{attribute 'pack_mode' := '1'} 
// ------------------------------------------------------------------------- 
//  SRCI Robot Library                                                
// ------------------------------------------------------------------------- 
//                                                                           
//  Object:      CalculateCartesianPositionParCmd                                       
//  Author:      Thorsten Brach                                                
//  Date:        2024-06-05
//
//  Description:                                              
//   
//                                                                           
//  Copyright: 
//    (C) 2024 Thorsten Brach. All rights reserved                                                                                                                                            
//             Licensed under the MIT License.
//                                                                           
//  Disclaimer:                                                                           
//    This project is provided without any guarantee and can be used for   
//    private and commercial purposes. Any use is at the user’s 
//    own risk and responsibility.
//
// -------------------------------------------------------------------------
TYPE CalculateCartesianPositionParCmd :
STRUCT
  /// Index of initial frame
  /// • 0: WCS (default)
  /// • 1..254: User frames
  FrameNo            : USINT;
  /// Index of target frame
  /// • 0: WCS (default)
  /// • 1..254: User frames
  TargetFrameNo      : USINT;  
  /// Robot cartesian position.
  CartesianPosition  : RobotCartesianPosition;
END_STRUCT
END_TYPE

{attribute 'pack_mode' := '1'} 
// ------------------------------------------------------------------------- 
//  SRCI Robot Library                                                
// ------------------------------------------------------------------------- 
//                                                                           
//  Object:      CalculateCartesianPositionRecvData                                       
//  Author:      Thorsten Brach                                                
//  Date:        2024-06-05
//
//  Description:                                              
//   
//                                                                           
//  Copyright: 
//    (C) 2024 Thorsten Brach. All rights reserved                                                                                                                                            
//             Licensed under the MIT License.
//                                                                           
//  Disclaimer:                                                                           
//    This project is provided without any guarantee and can be used for   
//    private and commercial purposes. Any use is at the user’s 
//    own risk and responsibility.
//
// -------------------------------------------------------------------------
TYPE CalculateCartesianPositionRecvData EXTENDS RspHeader :
STRUCT
  /// Index of target tool
  /// • 0: Flange (default)
  /// • 1..254: Tool frames
  TargetToolNoReturn       : USINT;
  /// Index of target frame
  /// •      0: WCS
  /// • 1..254: User frames
  TargetFrameNoReturn      : USINT;
  /// Calculated cartesian position
  CartesianPositionReturn  : RobotCartesianPosition;
END_STRUCT
END_TYPE

{attribute 'pack_mode' := '1'}
// ------------------------------------------------------------------------- 
//  SRCI Robot Library                                                
// ------------------------------------------------------------------------- 
//                                                                           
//  Object:      CalculateCartesianPositionSendData                                       
//  Author:      Thorsten Brach                                                
//  Date:        2024-06-05
//
//  Description:                                              
//   
//                                                                           
//  Copyright: 
//    (C) 2024 Thorsten Brach. All rights reserved                                                                                                                                            
//             Licensed under the MIT License.
//                                                                           
//  Disclaimer:                                                                           
//    This project is provided without any guarantee and can be used for   
//    private and commercial purposes. Any use is at the user’s 
//    own risk and responsibility.
//
// -------------------------------------------------------------------------
TYPE CalculateCartesianPositionSendData EXTENDS CmdHeader:   
STRUCT
  /// Index of source frame
  /// • 0: WCS (default)
  /// • 1..254: User frames
  FrameNo           : USINT;
  /// Index of target frame
  /// • 0: WCS (default)
  /// • 1..254: User frames
  TargetFrameNo     : USINT;
  /// Robot cartesian position.
  CartesianPosition : RobotCartesianPosition;
END_STRUCT
END_TYPE

{attribute 'pack_mode' := '1'} 
// ------------------------------------------------------------------------- 
//  SRCI Robot Library                                                
// ------------------------------------------------------------------------- 
//                                                                           
//  Object:      CalculateForwardKinematicOutCmd                                       
//  Author:      Thorsten Brach                                                
//  Date:        2024-06-05
//
//  Description:                                              
//   
//                                                                           
//  Copyright: 
//    (C) 2024 Thorsten Brach. All rights reserved                                                                                                                                            
//             Licensed under the MIT License.
//                                                                           
//  Disclaimer:                                                                           
//    This project is provided without any guarantee and can be used for   
//    private and commercial purposes. Any use is at the user’s 
//    own risk and responsibility.
//
// -------------------------------------------------------------------------
TYPE CalculateForwardKinematicOutCmd :
STRUCT
  /// Index of target tool
  /// • 0: Flange (default)
  /// • 1..254: Tool frames
  TargetToolNoReturn : USINT;
  /// Index of target frame
  /// •      0: WCS
  /// • 1..254: User frames
  TargetFrameNoReturn: USINT;
  /// Calculated cartesian position
  CartesianPosition  : RobotCartesianPosition;
END_STRUCT
END_TYPE

{attribute 'pack_mode' := '1'} 
// ------------------------------------------------------------------------- 
//  SRCI Robot Library                                                
// ------------------------------------------------------------------------- 
//                                                                           
//  Object:      CalculateForwardKinematicParCmd                                       
//  Author:      Thorsten Brach                                                
//  Date:        2024-06-05
//
//  Description:                                              
//   
//                                                                           
//  Copyright: 
//    (C) 2024 Thorsten Brach. All rights reserved                                                                                                                                            
//             Licensed under the MIT License.
//                                                                           
//  Disclaimer:                                                                           
//    This project is provided without any guarantee and can be used for   
//    private and commercial purposes. Any use is at the user’s 
//    own risk and responsibility.
//
// -------------------------------------------------------------------------
TYPE CalculateForwardKinematicParCmd :
STRUCT
  /// Index of target tool
  /// • 0: Flange (default)
  /// • 1..254: Tool frames
  ToolNo             : USINT;
  /// Index of target frame
  /// • 0: WCS (default)
  /// • 1..254: User frames
  FrameNo            : USINT;
  /// Calculate joint position
  JointPosition      : RobotJointPosition;
END_STRUCT
END_TYPE

{attribute 'pack_mode' := '1'} 
// ------------------------------------------------------------------------- 
//  SRCI Robot Library                                                
// ------------------------------------------------------------------------- 
//                                                                           
//  Object:      CalculateForwardKinematicRecvData                                       
//  Author:      Thorsten Brach                                                
//  Date:        2024-06-05
//
//  Description:                                              
//   
//                                                                           
//  Copyright: 
//    (C) 2024 Thorsten Brach. All rights reserved                                                                                                                                            
//             Licensed under the MIT License.
//                                                                           
//  Disclaimer:                                                                           
//    This project is provided without any guarantee and can be used for   
//    private and commercial purposes. Any use is at the user’s 
//    own risk and responsibility.
//
// -------------------------------------------------------------------------
TYPE CalculateForwardKinematicRecvData EXTENDS RspHeader :
STRUCT
  /// Index of target tool
  /// • 0: Flange (default)
  /// • 1..254: Tool frames
  TargetToolNoReturn       : USINT;
  /// Index of target frame
  /// •      0: WCS
  /// • 1..254: User frames
  TargetFrameNoReturn      : USINT;
  /// Calculated cartesian position
  CartesianPosition        : RobotCartesianPosition;
END_STRUCT
END_TYPE

{attribute 'pack_mode' := '1'}
// ------------------------------------------------------------------------- 
//  SRCI Robot Library                                                
// ------------------------------------------------------------------------- 
//                                                                           
//  Object:      CalculateForwardKinematicSendData                                       
//  Author:      Thorsten Brach                                                
//  Date:        2024-06-05
//
//  Description:                                              
//   
//                                                                           
//  Copyright: 
//    (C) 2024 Thorsten Brach. All rights reserved                                                                                                                                            
//             Licensed under the MIT License.
//                                                                           
//  Disclaimer:                                                                           
//    This project is provided without any guarantee and can be used for   
//    private and commercial purposes. Any use is at the user’s 
//    own risk and responsibility.
//
// -------------------------------------------------------------------------
TYPE CalculateForwardKinematicSendData EXTENDS CmdHeader:   
STRUCT
  /// Index of target tool
  /// • 0: Flange (default)
  /// • 1..254: Tool frames
  ToolNo        : USINT;
  /// Index of target frame
  /// • 0: WCS (default)
  /// • 1..254: User frames
  FrameNo        : USINT;
  /// Calculated joint position
  JointPosition  : RobotJointPosition;
END_STRUCT
END_TYPE

{attribute 'pack_mode' := '1'} 
// ------------------------------------------------------------------------- 
//  SRCI Robot Library                                                
// ------------------------------------------------------------------------- 
//                                                                           
//  Object:      CalculateFrameOutCmd                                       
//  Author:      Thorsten Brach                                                
//  Date:        2024-06-09
//
//  Description:                                              
//   
//                                                                           
//  Copyright: 
//    (C) 2024 Thorsten Brach. All rights reserved                                                                                                                                            
//             Licensed under the MIT License.
//                                                                           
//  Disclaimer:                                                                           
//    This project is provided without any guarantee and can be used for   
//    private and commercial purposes. Any use is at the user’s 
//    own risk and responsibility.
//
// -------------------------------------------------------------------------
TYPE CalculateFrameOutCmd :
STRUCT
  /// Date
  IEC_Date       : IEC_DATE;
  /// Time
  IEC_TIME       : IEC_TIME;
  /// Index of frame on which the calculated frame is depending
  /// •      0: WCS (default)
  /// • 1..254: User frames
  ReferenceFrame : USINT;
  /// Position
  Position       : RobotCartesianPositionBase;
END_STRUCT
END_TYPE

{attribute 'pack_mode' := '1'} 
// ------------------------------------------------------------------------- 
//  SRCI Robot Library                                                
// ------------------------------------------------------------------------- 
//                                                                           
//  Object:      CalculateFrameParCmd                                       
//  Author:      Thorsten Brach                                                
//  Date:        2024-06-09
//
//  Description:                                              
//   
//                                                                           
//  Copyright: 
//    (C) 2024 Thorsten Brach. All rights reserved                                                                                                                                            
//             Licensed under the MIT License.
//                                                                           
//  Disclaimer:                                                                           
//    This project is provided without any guarantee and can be used for   
//    private and commercial purposes. Any use is at the user’s 
//    own risk and responsibility.
//
// -------------------------------------------------------------------------
TYPE CalculateFrameParCmd :
STRUCT
  /// Define which method should be used to calculate the tool frame
  Mode               : FrameCalculationMode;
  /// Index of target frame
  /// • 0: WCS (default)
  /// • 1..254: User frames
  FrameNo            : USINT;  
  /// Cartesian position in the positive direction of the  X-Axis of the calculated frame coordinate system relative to the given frame
  Position_X         : RobotCartesianPosition;
  /// Cartesian position in the XY-plane of the calculated frame coordinate system relative to the given frame.
  Position_XY        : RobotCartesianPosition;
  /// Cartesian position of the origin of the calculated frame coordinate system relative to the given frame.
  Origin             : RobotCartesianPosition;
  /// Cartesian position of the postponement of the origin of the calculated frame coordinate system relative to the given frame.
  /// Auxiliary position if the origin of the can’t be reached by the robot, i.e. because it is inside an object.
  OriginShift        : RobotCartesianPosition;
  /// Index of frame on which the calculated frame is depending
  /// •      0: WCS (default)
  /// • 1..254: User frames
  ReferenceFrame     : USINT;
END_STRUCT
END_TYPE

{attribute 'pack_mode' := '1'} 
// ------------------------------------------------------------------------- 
//  SRCI Robot Library                                                
// ------------------------------------------------------------------------- 
//                                                                           
//  Object:      CalculateFrameRecvData                                       
//  Author:      Thorsten Brach                                                
//  Date:        2024-06-09
//
//  Description:                                              
//   
//                                                                           
//  Copyright: 
//    (C) 2024 Thorsten Brach. All rights reserved                                                                                                                                            
//             Licensed under the MIT License.
//                                                                           
//  Disclaimer:                                                                           
//    This project is provided without any guarantee and can be used for   
//    private and commercial purposes. Any use is at the user’s 
//    own risk and responsibility.
//
// -------------------------------------------------------------------------
TYPE CalculateFrameRecvData EXTENDS RspHeader :
STRUCT
  /// Date
  IEC_Date       : IEC_DATE;
  /// Time
  IEC_TIME       : IEC_TIME;
  /// Index of frame on which the calculated frame is depending
  /// •      0: WCS (default)
  /// • 1..254: User frames
  ReferenceFrame : USINT;
  /// Reserve
  Reserve        : BYTE;
  /// Position
  Position       : RobotCartesianPositionBase;
END_STRUCT
END_TYPE

{attribute 'pack_mode' := '1'}
// ------------------------------------------------------------------------- 
//  SRCI Robot Library                                                
// ------------------------------------------------------------------------- 
//                                                                           
//  Object:      CalculateFrameSendData                                       
//  Author:      Thorsten Brach                                                
//  Date:        2024-06-09
//
//  Description:                                              
//   
//                                                                           
//  Copyright: 
//    (C) 2024 Thorsten Brach. All rights reserved                                                                                                                                            
//             Licensed under the MIT License.
//                                                                           
//  Disclaimer:                                                                           
//    This project is provided without any guarantee and can be used for   
//    private and commercial purposes. Any use is at the user’s 
//    own risk and responsibility.
//
// -------------------------------------------------------------------------
TYPE CalculateFrameSendData EXTENDS CmdHeader:   
STRUCT
  /// Incremented with each position of the input parameter "PositionsArray" sent from the PLC to the RC.
  /// Default: 0
  DataIndex          : USINT;
  
  /// Set TRUE by the client, when according to the user selected "Mode" the final position of the input parameter "PositionsArray" is sent to the RC.
  /// Default: FALSE
  DataComplete       : BYTE;
  ///
  Reserve            : BYTE;
  /// Index of target frame
  /// • 0: WCS (default)
  /// • 1..254: User frames
  FrameNo            : USINT;
  /// Index of frame on which the calculated frame is depending
  /// •      0: WCS (default)
  /// • 1..254: User frames
  ReferenceFrame     : USINT;
  /// Define which method should be used to calculate the frame coordinate system: M
  /// • 0: Three-Point-Method (default) O
  /// • 1: Four-Point-Method O
  /// • 2: One-Point-Method
  Mode               : SINT;  
  /// Cartesian position
  Position           : RobotCartesianPosition;  
END_STRUCT
END_TYPE

{attribute 'pack_mode' := '1'} 
// ------------------------------------------------------------------------- 
//  SRCI Robot Library                                                
// ------------------------------------------------------------------------- 
//                                                                           
//  Object:      CalculateInverseKinematicOutCmd                                       
//  Author:      Thorsten Brach                                                
//  Date:        2024-06-09
//
//  Description:                                              
//   
//                                                                           
//  Copyright: 
//    (C) 2024 Thorsten Brach. All rights reserved                                                                                                                                                                                                               
//             Licensed under the MIT License.
//                                                                           
//  Disclaimer:                                                                           
//    This project is provided without any guarantee and can be used for   
//    private and commercial purposes. Any use is at the user’s 
//    own risk and responsibility.
//
// -------------------------------------------------------------------------
TYPE CalculateInverseKinematicOutCmd :
STRUCT
  /// Calculated robot joint position
  JointPosition      : RobotJointPosition;  
END_STRUCT
END_TYPE

{attribute 'pack_mode' := '1'} 
// ------------------------------------------------------------------------- 
//  SRCI Robot Library                                                
// ------------------------------------------------------------------------- 
//                                                                           
//  Object:      CalculateInverseKinematicParCmd                                       
//  Author:      Thorsten Brach                                                
//  Date:        2024-06-09
//
//  Description:                                              
//   
//                                                                           
//  Copyright: 
//    (C) 2024 Thorsten Brach. All rights reserved                                                                                                                                      
//             Licensed under the MIT License.
//                                                                           
//  Disclaimer:                                                                           
//    This project is provided without any guarantee and can be used for   
//    private and commercial purposes. Any use is at the user’s 
//    own risk and responsibility.
//
// -------------------------------------------------------------------------
TYPE CalculateInverseKinematicParCmd :
STRUCT
  /// cartesian position
  CartesianPosition  : RobotCartesianPosition;
  /// Index of target tool
  /// • 0: Flange (default)
  /// • 1..254: Tool frames
  ToolNo             : USINT;
  /// Index of target frame
  /// • 0: WCS (default)
  /// • 1..254: User frames
  FrameNo            : USINT;  
END_STRUCT
END_TYPE

{attribute 'pack_mode' := '1'} 
// ------------------------------------------------------------------------- 
//  SRCI Robot Library                                                
// ------------------------------------------------------------------------- 
//                                                                           
//  Object:      CalculateInverseKinematicRecvData                                       
//  Author:      Thorsten Brach                                                
//  Date:        2024-06-09
//
//  Description:                                              
//   
//                                                                           
//  Copyright: 
//    (C) 2024 Thorsten Brach. All rights reserved                                                                                                                                            
//             Licensed under the MIT License.
//                                                                           
//  Disclaimer:                                                                           
//    This project is provided without any guarantee and can be used for   
//    private and commercial purposes. Any use is at the user’s 
//    own risk and responsibility.
//
// -------------------------------------------------------------------------
TYPE CalculateInverseKinematicRecvData EXTENDS RspHeader :
STRUCT
  /// Calculated robot joint position
  JointPosition      : RobotJointPosition;  
END_STRUCT
END_TYPE

{attribute 'pack_mode' := '1'}
// ------------------------------------------------------------------------- 
//  SRCI Robot Library                                                
// ------------------------------------------------------------------------- 
//                                                                           
//  Object:      CalculateInverseKinematicSendData                                       
//  Author:      Thorsten Brach                                                
//  Date:        2024-06-09
//
//  Description:                                              
//   
//                                                                           
//  Copyright: 
//    (C) 2024 Thorsten Brach. All rights reserved                                                                                                                                            
//             Licensed under the MIT License.
//                                                                           
//  Disclaimer:                                                                           
//    This project is provided without any guarantee and can be used for   
//    private and commercial purposes. Any use is at the user’s 
//    own risk and responsibility.
//
// -------------------------------------------------------------------------
TYPE CalculateInverseKinematicSendData EXTENDS CmdHeader:   
STRUCT
  /// cartesian position
  CartesianPosition  : RobotCartesianPosition;
  /// Index of target tool
  /// • 0: Flange (default)
  /// • 1..254: Tool frames
  ToolNo             : USINT;
  /// Index of target frame
  /// • 0: WCS (default)
  /// • 1..254: User frames
  FrameNo            : USINT;  
END_STRUCT
END_TYPE

{attribute 'pack_mode' := '1'} 
// ------------------------------------------------------------------------- 
//  SRCI Robot Library                                                
// ------------------------------------------------------------------------- 
//                                                                           
//  Object:      CalculateToolOutCmd                                       
//  Author:      Thorsten Brach                                                
//  Date:        2024-06-09
//
//  Description:                                              
//   
//                                                                           
//  Copyright: 
//    (C) 2024 Thorsten Brach. All rights reserved                                                                                                                                                                                                               
//             Licensed under the MIT License.
//                                                                           
//  Disclaimer:                                                                           
//    This project is provided without any guarantee and can be used for   
//    private and commercial purposes. Any use is at the user’s 
//    own risk and responsibility.
//
// -------------------------------------------------------------------------
TYPE CalculateToolOutCmd :
STRUCT
  /// Tool data
  ToolData           : ToolData;
  /// Maximum error of deviation of the TCP position
  /// from the fix point in world coordinate system
  /// If not supported: • -1
  TCPMaxError       : REAL;
  /// Average error of TCP position from the fix point  in world coordinate system
  /// If not supported: • -1 
  TCPMeanError      : REAL;
END_STRUCT
END_TYPE

{attribute 'pack_mode' := '1'} 
// ------------------------------------------------------------------------- 
//  SRCI Robot Library                                                
// ------------------------------------------------------------------------- 
//                                                                           
//  Object:      CalculateToolParCmd                                       
//  Author:      Thorsten Brach                                                
//  Date:        2024-06-09
//
//  Description:                                              
//   
//                                                                           
//  Copyright: 
//    (C) 2024 Thorsten Brach. All rights reserved                                                                                                                                      
//             Licensed under the MIT License.
//                                                                           
//  Disclaimer:                                                                           
//    This project is provided without any guarantee and can be used for   
//    private and commercial purposes. Any use is at the user’s 
//    own risk and responsibility.
//
// -------------------------------------------------------------------------
TYPE CalculateToolParCmd :
STRUCT
  /// Define which method should be used to calculate the tool frame
  Mode               : ToolCalculationMode;
  /// Index of target tool
  /// • 0: Flange (default)
  /// • 1..254: Tool frames
  ToolNo             : USINT;
  /// Index of target frame
  /// • 0: WCS (default)
  /// • 1..254: User frames
  FrameNo            : USINT;  
  /// • True: Tool fixed
  /// • False: Tool on flange (default)
  ExternalTCP        : BOOL;
  /// Positions in cartesian coordinates for the tool frame calculation.
  PositionsArray     : ARRAY[0..5] OF RobotCartesianPosition;
END_STRUCT
END_TYPE

{attribute 'pack_mode' := '1'} 
// ------------------------------------------------------------------------- 
//  SRCI Robot Library                                                
// ------------------------------------------------------------------------- 
//                                                                           
//  Object:      CalculateToolRecvData                                       
//  Author:      Thorsten Brach                                                
//  Date:        2024-06-09
//
//  Description:                                              
//   
//                                                                           
//  Copyright: 
//    (C) 2024 Thorsten Brach. All rights reserved                                                                                                                                            
//             Licensed under the MIT License.
//                                                                           
//  Disclaimer:                                                                           
//    This project is provided without any guarantee and can be used for   
//    private and commercial purposes. Any use is at the user’s 
//    own risk and responsibility.
//
// -------------------------------------------------------------------------
TYPE CalculateToolRecvData EXTENDS RspHeader :
STRUCT
  /// Maximum error of deviation of the TCP position
  /// from the fix point in world coordinate system
  /// If not supported: • -1
  TCPMaxError       : REAL;
  /// Average error of TCP position from the fix point  in world coordinate system
  /// If not supported: • -1 
  TCPMeanError      : REAL;
  /// Tool data
  ToolData           : ToolData;
END_STRUCT
END_TYPE

{attribute 'pack_mode' := '1'}
// ------------------------------------------------------------------------- 
//  SRCI Robot Library                                                
// ------------------------------------------------------------------------- 
//                                                                           
//  Object:      CalculateToolSendData                                       
//  Author:      Thorsten Brach                                                
//  Date:        2024-06-09
//
//  Description:                                              
//   
//                                                                           
//  Copyright: 
//    (C) 2024 Thorsten Brach. All rights reserved                                                                                                                                            
//             Licensed under the MIT License.
//                                                                           
//  Disclaimer:                                                                           
//    This project is provided without any guarantee and can be used for   
//    private and commercial purposes. Any use is at the user’s 
//    own risk and responsibility.
//
// -------------------------------------------------------------------------
TYPE CalculateToolSendData EXTENDS CmdHeader:   
STRUCT
  DataIndex    : USINT;
  ///
  DataComplete : BYTE;
  /// Index of target tool
  /// • 0: Flange (default)
  /// • 1..254: Tool frames
  ToolNo       : USINT;
  /// Index of target frame
  /// • 0: WCS (default)
  /// • 1..254: User frames
  FrameNo      : USINT;    
  /// Define which method should be used to calculate the tool frame
  Mode         : ToolCalculationMode;
  /// • True: Tool fixed
  /// • False: Tool on flange (default)
  ExternalTCP  : USINT;
  /// Positions in cartesian coordinates for the tool frame calculation.
  Position     : RobotCartesianPosition;
END_STRUCT
END_TYPE

{attribute 'pack_mode' := '1'} 
// ------------------------------------------------------------------------- 
//  SRCI Robot Library                                                
// ------------------------------------------------------------------------- 
//                                                                           
//  Object:      LoadMeasurementAutomaticOutCmd                                       
//  Author:      Thorsten Brach                                                
//  Date:        2024-06-20
//
//  Description:                                              
//   
//                                                                           
//  Copyright: 
//    (C) 2024 Thorsten Brach. All rights reserved                                                                                                                                            
//             Licensed under the MIT License.
//                                                                           
//  Disclaimer:                                                                           
//    This project is provided without any guarantee and can be used for   
//    private and commercial purposes. Any use is at the user’s 
//    own risk and responsibility.
//
// -------------------------------------------------------------------------
TYPE LoadMeasurementAutomaticOutCmd :
STRUCT
  /// FB is returning a unique ID for the cal led measurement.
  MeasuringID       : UINT;
  /// Measured load data (see chapter 5.5.6.4)
  LoadData          : LoadData;  
  /// Load data available
  LoadDataAvailable : BOOL;
END_STRUCT
END_TYPE

{attribute 'pack_mode' := '1'} 
// ------------------------------------------------------------------------- 
//  SRCI Robot Library                                                
// ------------------------------------------------------------------------- 
//                                                                           
//  Object:      LoadMeasurementAutomaticParCmd                                       
//  Author:      Thorsten Brach                                                
//  Date:        2024-06-20
//
//  Description:                                              
//   
//                                                                           
//  Copyright: 
//    (C) 2024 Thorsten Brach. All rights reserved                                                                                                                                            
//             Licensed under the MIT License.
//                                                                           
//  Disclaimer:                                                                           
//    This project is provided without any guarantee and can be used for   
//    private and commercial purposes. Any use is at the user’s 
//    own risk and responsibility.
//
// -------------------------------------------------------------------------
TYPE LoadMeasurementAutomaticParCmd :
STRUCT
  /// Define which method should be used to measure the load data
  Mode               : LoadMeasurementMode;
  /// Define which mass is expected as a result of the load measurement
  Mass               : REAL;
  /// Define the area for the allowed motion of the Joint 3. 
  /// The order of the two limit values does not matter. 
  /// Only considered with "Mode" = 0, 2.
  Area_J3            : ARRAY[0..1] OF REAL;
  /// Define the area for the allowed motion of the Joint 4. 
  /// The order of the two limit values does not matter. 
  /// Only considered with "Mode" = 0, 2.
  Area_J4            : ARRAY[0..1] OF REAL;
  /// Define the area for the allowed motion of the Joint 5. 
  /// The order of the two limit values does not matter. 
  /// Only considered with "Mode" = 0, 2.
  Area_J5            : ARRAY[0..1] OF REAL;
  /// Define the area for the allowed motion of the Joint 6. 
  /// The order of the two limit values does not matter. 
  /// Only considered with "Mode" = 0, 2.
  Area_J6            : ARRAY[0..1] OF REAL;
  /// Define the first position for the load measurement.
  /// Only considered with "Mode" = 0, 1.
  Position_1         : RobotJointPosition;
  /// Define the second position for the load measurement.
  /// Only considered with "Mode" = 3.
  Position_2         : RobotJointPosition;
  /// Define the configuration angle for the load measurement.
  /// Only considered with "Mode" = 1.
  ConfigurationAngle : REAL;
END_STRUCT
END_TYPE

{attribute 'pack_mode' := '1'} 
// ------------------------------------------------------------------------- 
//  SRCI Robot Library                                                
// ------------------------------------------------------------------------- 
//                                                                           
//  Object:      LoadMeasurementAutomaticRecvData                                       
//  Author:      Thorsten Brach                                                
//  Date:        2024-06-20
//
//  Description:                                              
//   
//                                                                           
//  Copyright: 
//    (C) 2024 Thorsten Brach. All rights reserved                                                                                                                                            
//             Licensed under the MIT License.
//                                                                           
//  Disclaimer:                                                                           
//    This project is provided without any guarantee and can be used for   
//    private and commercial purposes. Any use is at the user’s 
//    own risk and responsibility.
//
// -------------------------------------------------------------------------
TYPE LoadMeasurementAutomaticRecvData EXTENDS RspHeader :
STRUCT
    /// FB is returning a unique ID for the cal led measurement.
  MeasuringID       : UINT;
  /// Measured load data (see chapter 5.5.6.4)
  LoadData          : LoadData;  
  /// Load data available
  LoadDataAvailable : BOOL;
END_STRUCT
END_TYPE

{attribute 'pack_mode' := '1'}
// ------------------------------------------------------------------------- 
//  SRCI Robot Library                                                
// ------------------------------------------------------------------------- 
//                                                                           
//  Object:      LoadMeasurementAutomaticSendData                                       
//  Author:      Thorsten Brach                                                
//  Date:        2024-06-20
//
//  Description:                                              
//   
//                                                                           
//  Copyright: 
//    (C) 2024 Thorsten Brach. All rights reserved                                                                                                                                            
//             Licensed under the MIT License.
//                                                                           
//  Disclaimer:                                                                           
//    This project is provided without any guarantee and can be used for   
//    private and commercial purposes. Any use is at the user’s 
//    own risk and responsibility.
//
// -------------------------------------------------------------------------
TYPE LoadMeasurementAutomaticSendData EXTENDS CmdHeader:   
STRUCT
    /// Define which mass is expected as a result of the load measurement
  Mass               : REAL;
  /// Define which method should be used to measure the load data
  Mode               : LoadMeasurementMode;
  /// Reserved
  Reserved           : BYTE;
  /// Define the area for the allowed motion of the Joint 3. 
  /// The order of the two limit values does not matter. 
  /// Only considered with "Mode" = 0, 2.
  Area_J3            : ARRAY[0..1] OF REAL;
  /// Define the area for the allowed motion of the Joint 4. 
  /// The order of the two limit values does not matter. 
  /// Only considered with "Mode" = 0, 2.
  Area_J4            : ARRAY[0..1] OF REAL;
  /// Define the area for the allowed motion of the Joint 5. 
  /// The order of the two limit values does not matter. 
  /// Only considered with "Mode" = 0, 2.
  Area_J5            : ARRAY[0..1] OF REAL;
  /// Define the area for the allowed motion of the Joint 6. 
  /// The order of the two limit values does not matter. 
  /// Only considered with "Mode" = 0, 2.
  Area_J6            : ARRAY[0..1] OF REAL;
  /// Define the configuration angle for the load measurement.
  /// Only considered with "Mode" = 1.
  ConfigurationAngle : REAL;
  /// Define the first position for the load measurement.
  /// Only considered with "Mode" = 0, 1.
  Position_1         : RobotJointPosition;
  /// Define the second position for the load measurement.
  /// Only considered with "Mode" = 3.
  Position_2         : RobotJointPosition;
END_STRUCT
END_TYPE

{attribute 'pack_mode' := '1'} 
// ------------------------------------------------------------------------- 
//  SRCI Robot Library                                                
// ------------------------------------------------------------------------- 
//                                                                           
//  Object:      LoadMeasurementSequentialOutCmd                                       
//  Author:      Thorsten Brach                                                
//  Date:        2024-06-20
//
//  Description:                                              
//   
//                                                                           
//  Copyright: 
//    (C) 2024 Thorsten Brach. All rights reserved                                                                                                                                            
//             Licensed under the MIT License.
//                                                                           
//  Disclaimer:                                                                           
//    This project is provided without any guarantee and can be used for   
//    private and commercial purposes. Any use is at the user’s 
//    own risk and responsibility.
//
// -------------------------------------------------------------------------
TYPE LoadMeasurementSequentialOutCmd :
STRUCT
  /// FB is returning a unique ID for the cal led measurement.
  MeasuringID        : UINT;
  /// Measured load data (see chapter 5.5.6.4)
  LoadData           : LoadData;
  /// Load data available
  LoadDataAvailable : BOOL;
END_STRUCT
END_TYPE

{attribute 'pack_mode' := '1'} 
// ------------------------------------------------------------------------- 
//  SRCI Robot Library                                                
// ------------------------------------------------------------------------- 
//                                                                           
//  Object:      LoadMeasurementSequentialParCmd                                       
//  Author:      Thorsten Brach                                                
//  Date:        2024-06-20
//
//  Description:                                              
//   
//                                                                           
//  Copyright: 
//    (C) 2024 Thorsten Brach. All rights reserved                                                                                                                                            
//             Licensed under the MIT License.
//                                                                           
//  Disclaimer:                                                                           
//    This project is provided without any guarantee and can be used for   
//    private and commercial purposes. Any use is at the user’s 
//    own risk and responsibility.
//
// -------------------------------------------------------------------------
TYPE LoadMeasurementSequentialParCmd :
STRUCT
  /// Define which step of the load estimation should be executed:
  Mode               : LoadMeasurementSteps;
  /// Define which mass is expected as a result of the load measurement
  Mass               : REAL;
END_STRUCT
END_TYPE

{attribute 'pack_mode' := '1'} 
// ------------------------------------------------------------------------- 
//  SRCI Robot Library                                                
// ------------------------------------------------------------------------- 
//                                                                           
//  Object:      LoadMeasurementSequentialRecvData                                       
//  Author:      Thorsten Brach                                                
//  Date:        2024-06-20
//
//  Description:                                              
//   
//                                                                           
//  Copyright: 
//    (C) 2024 Thorsten Brach. All rights reserved                                                                                                                                            
//             Licensed under the MIT License.
//                                                                           
//  Disclaimer:                                                                           
//    This project is provided without any guarantee and can be used for   
//    private and commercial purposes. Any use is at the user’s 
//    own risk and responsibility.
//
// -------------------------------------------------------------------------
TYPE LoadMeasurementSequentialRecvData EXTENDS RspHeader :
STRUCT
  /// FB is returning a unique ID for the cal led measurement.
  MeasuringID       : UINT;
  /// Measured load data (see chapter 5.5.6.4)
  LoadData          : LoadData;  
  /// Load data available
  LoadDataAvailable : BOOL;
END_STRUCT
END_TYPE

{attribute 'pack_mode' := '1'}
// ------------------------------------------------------------------------- 
//  SRCI Robot Library                                                
// ------------------------------------------------------------------------- 
//                                                                           
//  Object:      LoadMeasurementSequentialSendData                                       
//  Author:      Thorsten Brach                                                
//  Date:        2024-06-20
//
//  Description:                                              
//   
//                                                                           
//  Copyright: 
//    (C) 2024 Thorsten Brach. All rights reserved                                                                                                                                            
//             Licensed under the MIT License.
//                                                                           
//  Disclaimer:                                                                           
//    This project is provided without any guarantee and can be used for   
//    private and commercial purposes. Any use is at the user’s 
//    own risk and responsibility.
//
// -------------------------------------------------------------------------
TYPE LoadMeasurementSequentialSendData EXTENDS CmdHeader:   
STRUCT
    /// Define which mass is expected as a result of the load measurement
  Mass               : REAL;
  /// Define which step of the load estimation should be executed:
  Mode               : LoadMeasurementSteps;
END_STRUCT
END_TYPE

{attribute 'pack_mode' := '1'} 
// ------------------------------------------------------------------------- 
//  SRCI Robot Library                                                
// ------------------------------------------------------------------------- 
//                                                                           
//  Object:      ActivateConveyorTrackingOutCmd                                       
//  Author:      Thorsten Brach                                                
//  Date:        2024-06-11
//
//  Description:                                              
//   
//                                                                           
//  Copyright: 
//    (C) 2024 Thorsten Brach. All rights reserved                                                                                                                                                                                                               
//             Licensed under the MIT License.
//                                                                           
//  Disclaimer:                                                                           
//    This project is provided without any guarantee and can be used for   
//    private and commercial purposes. Any use is at the user’s 
//    own risk and responsibility.
//
// -------------------------------------------------------------------------
TYPE ActivateConveyorTrackingOutCmd :
STRUCT
  /// Current status of "ConveyorTracking" according to Table 6-432
  TrackingStatus     : TrackingStatus;
  /// Relates to "ConnectionMode" 1 – "RC connected": Traveled distance of assigned conveyor since ConveyorTracking has been activated (offset)
  RCEncoderValue     : REAL;
END_STRUCT
END_TYPE

{attribute 'pack_mode' := '1'} 
// ------------------------------------------------------------------------- 
//  SRCI Robot Library                                                
// ------------------------------------------------------------------------- 
//                                                                           
//  Object:      ActivateConveyorTrackingParCmd                                       
//  Author:      Thorsten Brach                                                
//  Date:        2024-06-11
//
//  Description:                                              
//   
//                                                                           
//  Copyright: 
//    (C) 2024 Thorsten Brach. All rights reserved                                                                                                                                      
//             Licensed under the MIT License.
//                                                                           
//  Disclaimer:                                                                           
//    This project is provided without any guarantee and can be used for   
//    private and commercial purposes. Any use is at the user’s 
//    own risk and responsibility.
//
// -------------------------------------------------------------------------
TYPE ActivateConveyorTrackingParCmd :
STRUCT
  /// Index of assigned conveyor
  ConveyorNo         : SINT;
  /// Specifies encoder connection setup (at least one option must be supported)
  ConnectionMode     : ConnectionMode;
  /// Relates to "ConnectionMode" 1 – "PLC connected": Value of the encoder connected to the conveyor belt
  PLCEncoderValue    : REAL;
END_STRUCT
END_TYPE

{attribute 'pack_mode' := '1'} 
// ------------------------------------------------------------------------- 
//  SRCI Robot Library                                                
// ------------------------------------------------------------------------- 
//                                                                           
//  Object:      ActivateConveyorTrackingRecvData                                       
//  Author:      Thorsten Brach                                                
//  Date:        2024-06-11
//
//  Description:                                              
//   
//                                                                           
//  Copyright: 
//    (C) 2024 Thorsten Brach. All rights reserved                                                                                                                                            
//             Licensed under the MIT License.
//                                                                           
//  Disclaimer:                                                                           
//    This project is provided without any guarantee and can be used for   
//    private and commercial purposes. Any use is at the user’s 
//    own risk and responsibility.
//
// -------------------------------------------------------------------------
TYPE ActivateConveyorTrackingRecvData EXTENDS RspHeader :
STRUCT
  /// Maximum error of deviation of the TCP position
  /// from the fix point in world coordinate system
  /// If not supported: • -1
  TrackingStatus : TrackingStatus;
END_STRUCT
END_TYPE

{attribute 'pack_mode' := '1'}
// ------------------------------------------------------------------------- 
//  SRCI Robot Library                                                
// ------------------------------------------------------------------------- 
//                                                                           
//  Object:      ActivateConveyorTrackingSendData                                       
//  Author:      Thorsten Brach                                                
//  Date:        2024-06-11
//
//  Description:                                              
//   
//                                                                           
//  Copyright: 
//    (C) 2024 Thorsten Brach. All rights reserved                                                                                                                                            
//             Licensed under the MIT License.
//                                                                           
//  Disclaimer:                                                                           
//    This project is provided without any guarantee and can be used for   
//    private and commercial purposes. Any use is at the user’s 
//    own risk and responsibility.
//
// -------------------------------------------------------------------------
TYPE ActivateConveyorTrackingSendData EXTENDS CmdHeader:   
STRUCT
  /// Index of assigned conveyor
  ConveyorNo     : SINT;
  /// Specifies encoder connection setup (at least one option must be supported)
  ConnectionMode : SINT;
END_STRUCT
END_TYPE

{attribute 'pack_mode' := '1'} 
// ------------------------------------------------------------------------- 
//  SRCI Robot Library                                                
// ------------------------------------------------------------------------- 
//                                                                           
//  Object:      ConfigureConveyorOutCmd                                       
//  Author:      Thorsten Brach                                                
//  Date:        2024-06-11
//
//  Description:                                              
//   
//                                                                           
//  Copyright: 
//    (C) 2024 Thorsten Brach. All rights reserved                                                                                                                                                                                                               
//             Licensed under the MIT License.
//                                                                           
//  Disclaimer:                                                                           
//    This project is provided without any guarantee and can be used for   
//    private and commercial purposes. Any use is at the user’s 
//    own risk and responsibility.
//
// -------------------------------------------------------------------------
TYPE ConfigureConveyorOutCmd :
STRUCT
END_STRUCT
END_TYPE

{attribute 'pack_mode' := '1'} 
// ------------------------------------------------------------------------- 
//  SRCI Robot Library                                                
// ------------------------------------------------------------------------- 
//                                                                           
//  Object:      ConfigureConveyorParCmd                                       
//  Author:      Thorsten Brach                                                
//  Date:        2024-06-11
//
//  Description:                                              
//   
//                                                                           
//  Copyright: 
//    (C) 2024 Thorsten Brach. All rights reserved                                                                                                                                      
//             Licensed under the MIT License.
//                                                                           
//  Disclaimer:                                                                           
//    This project is provided without any guarantee and can be used for   
//    private and commercial purposes. Any use is at the user’s 
//    own risk and responsibility.
//
// -------------------------------------------------------------------------
TYPE ConfigureConveyorParCmd :
STRUCT
  /// Index of assigned conveyor
  ConveyorNo         : USINT;  
  ///Define the origin coordinate system of the conveyor belt, with the X-Axis pointing in the direction of the movement of the conveyor belt.
  ConveyorOrigin     : FrameData;
  /// Define the type of the conveyor
  ConveyorType       : ConveyorType;
  /// Relates to "ConveyorType" "Circular Tracking": Define the radius of the circular conveyor
  Radius             : REAL;
  /// Distance [mm] from the origin of the conveyor belt to the beginning of the "SyncInZone"
  StartDistance      : REAL;
  /// Distance [mm] from the origin of the conveyor belt to the end of the "SyncOutZone"
  EndDistance        : REAL;
  /// Define the length of the "SyncInZone"
  SyncInLength       : REAL;
  /// Define the length of the "SyncOutZone"
  SyncOutLength      : REAL;
END_STRUCT
END_TYPE

{attribute 'pack_mode' := '1'} 
// ------------------------------------------------------------------------- 
//  SRCI Robot Library                                                
// ------------------------------------------------------------------------- 
//                                                                           
//  Object:      ConfigureConveyorRecvData                                       
//  Author:      Thorsten Brach                                                
//  Date:        2024-06-11
//
//  Description:                                              
//   
//                                                                           
//  Copyright: 
//    (C) 2024 Thorsten Brach. All rights reserved                                                                                                                                            
//             Licensed under the MIT License.
//                                                                           
//  Disclaimer:                                                                           
//    This project is provided without any guarantee and can be used for   
//    private and commercial purposes. Any use is at the user’s 
//    own risk and responsibility.
//
// -------------------------------------------------------------------------
TYPE ConfigureConveyorRecvData EXTENDS RspHeader :
STRUCT
END_STRUCT
END_TYPE

{attribute 'pack_mode' := '1'}
// ------------------------------------------------------------------------- 
//  SRCI Robot Library                                                
// ------------------------------------------------------------------------- 
//                                                                           
//  Object:      ConfigureConveyorSendData                                       
//  Author:      Thorsten Brach                                                
//  Date:        2024-06-11
//
//  Description:                                              
//   
//                                                                           
//  Copyright: 
//    (C) 2024 Thorsten Brach. All rights reserved                                                                                                                                            
//             Licensed under the MIT License.
//                                                                           
//  Disclaimer:                                                                           
//    This project is provided without any guarantee and can be used for   
//    private and commercial purposes. Any use is at the user’s 
//    own risk and responsibility.
//
// -------------------------------------------------------------------------
TYPE ConfigureConveyorSendData EXTENDS CmdHeader:   
STRUCT
  ///Define the origin coordinate system of the conveyor belt, with the X-Axis pointing in the direction of the movement of the conveyor belt.
  ConveyorOrigin          : FrameData;
  /// ConveyorOrigin available
  ConveyorOriginAvailable : BOOL;
  /// Index of assigned conveyor
  ConveyorNo              : USINT;  
  /// Define the type of the conveyor
  ConveyorType            : ConveyorType;
  /// Relates to "ConveyorType" "Circular Tracking": Define the radius of the circular conveyor
  Radius                  : REAL;
  /// Distance [mm] from the origin of the conveyor belt to the beginning of the "SyncInZone"
  StartDistance           : REAL;
  /// Distance [mm] from the origin of the conveyor belt to the end of the "SyncOutZone"
  EndDistance             : REAL;
  /// Define the length of the "SyncInZone"
  SyncInLength            : REAL;
  /// Define the length of the "SyncOutZone"
  SyncOutLength           : REAL;
END_STRUCT
END_TYPE

{attribute 'pack_mode' := '1'} 
// ------------------------------------------------------------------------- 
//  SRCI Robot Library                                                
// ------------------------------------------------------------------------- 
//                                                                           
//  Object:      RedefineTrackingPosOutCmd                                       
//  Author:      Thorsten Brach                                                
//  Date:        2024-06-11
//
//  Description:                                              
//   
//                                                                           
//  Copyright: 
//    (C) 2024 Thorsten Brach. All rights reserved                                                                                                                                                                                                               
//             Licensed under the MIT License.
//                                                                           
//  Disclaimer:                                                                           
//    This project is provided without any guarantee and can be used for   
//    private and commercial purposes. Any use is at the user’s 
//    own risk and responsibility.
//
// -------------------------------------------------------------------------
TYPE RedefineTrackingPosOutCmd :
STRUCT
  /// Unique system-generated ID of the "Action" when the function is triggered.
  /// • >0: The "Action" is started by the trigger funcrion with identical FollowID.
  /// • <0: The "Action" is stopped by the trigger function with identical FollowID.
  /// For more information see chapter 5.5.12.4 EmitterID, ListenerID, FollowID and OriginID
  OriginID               : INT;
  /// Relates to ListenerID >0
  /// Number of successful trigger-based command invocations - For more information refer TO chapter 5.5.12.4
  InvocationCounter      : USINT;  
END_STRUCT
END_TYPE

{attribute 'pack_mode' := '1'} 
// ------------------------------------------------------------------------- 
//  SRCI Robot Library                                                
// ------------------------------------------------------------------------- 
//                                                                           
//  Object:      RedefineTrackingPosParCmd                                       
//  Author:      Thorsten Brach                                                
//  Date:        2024-06-11
//
//  Description:                                              
//   
//                                                                           
//  Copyright: 
//    (C) 2024 Thorsten Brach. All rights reserved                                                                                                                                      
//             Licensed under the MIT License.
//                                                                           
//  Disclaimer:                                                                           
//    This project is provided without any guarantee and can be used for   
//    private and commercial purposes. Any use is at the user’s 
//    own risk and responsibility.
//
// -------------------------------------------------------------------------
TYPE RedefineTrackingPosParCmd :
STRUCT
  /// Index of assigned conveyor
  ConveyorNo             : USINT;
  /// Relates to ListenerID = 0:
  /// Define initial work piece position relative to the conveyor belt origin:
  /// • Origin (X, Y, Z in mm)
  /// • Orientation (RX, RY, RZ in degree)
  /// For more information refer to chapter 5.5.14.
  InitObjectPosition     : ARRAY[0..5] OF REAL;
  /// Relates to ListenerID = 0:
  /// Travel distance of assigned UCS between work piece detection (InitObjectPosition) and execution of this command.
  TrackingOffset         : REAL;
  /// Relates to ListenerID >0
  /// Start index of real registers containing InitObjectPosition for trigger-based execution.
  StartIndexInitPosition : USINT;
  /// Define the index number of the UCS that is assigned to the conveyor by the function "ConveyorTracking".
  /// For more information refer to chapter 5.5.14.
  FrameNo                : USINT;
  /// Relates to ListenerID >0
  /// Index of real register containing TrackingOffset for trigger-based execution
  IndexTrackingOffset    : USINT;
  /// ID of associated trigger function:
  /// • 0: No Trigger (default): No trigger related behavior
  /// • >0: Trigger: o Start executing, when the trigger function with the identical EmitterID is triggered.
  /// Always positive.
  /// For more information, see chapter 5.5.12 Triggers
  ListenerID             :  SINT;
END_STRUCT
END_TYPE

{attribute 'pack_mode' := '1'} 
// ------------------------------------------------------------------------- 
//  SRCI Robot Library                                                
// ------------------------------------------------------------------------- 
//                                                                           
//  Object:      RedefineTrackingPosRecvData                                       
//  Author:      Thorsten Brach                                                
//  Date:        2024-06-11
//
//  Description:                                              
//   
//                                                                           
//  Copyright: 
//    (C) 2024 Thorsten Brach. All rights reserved                                                                                                                                            
//             Licensed under the MIT License.
//                                                                           
//  Disclaimer:                                                                           
//    This project is provided without any guarantee and can be used for   
//    private and commercial purposes. Any use is at the user’s 
//    own risk and responsibility.
//
// -------------------------------------------------------------------------
TYPE RedefineTrackingPosRecvData EXTENDS RspHeader :
STRUCT
  
  InvocationCounter : USINT;
  /// Reserve
  Reserved          : SINT;
  /// Unique system-generated ID of the "Action" when the function is triggered.
  /// • >0: The "Action" is started by the trigger funcrion with identical FollowID.
  /// • <0: The "Action" is stopped by the trigger function with identical FollowID.
  /// For more information see chapter 5.5.12.4 EmitterID, ListenerID, FollowID and OriginID
  OriginID          : INT;
END_STRUCT
END_TYPE

{attribute 'pack_mode' := '1'}
// ------------------------------------------------------------------------- 
//  SRCI Robot Library                                                
// ------------------------------------------------------------------------- 
//                                                                           
//  Object:      RedefineTrackingPosSendData                                       
//  Author:      Thorsten Brach                                                
//  Date:        2024-06-11
//
//  Description:                                              
//   
//                                                                           
//  Copyright: 
//    (C) 2024 Thorsten Brach. All rights reserved                                                                                                                                            
//             Licensed under the MIT License.
//                                                                           
//  Disclaimer:                                                                           
//    This project is provided without any guarantee and can be used for   
//    private and commercial purposes. Any use is at the user’s 
//    own risk and responsibility.
//
// -------------------------------------------------------------------------
TYPE RedefineTrackingPosSendData EXTENDS CmdHeader:   
STRUCT
  /// EmitterID
  EmitterID              : ARRAY[0..3] OF SINT;
  /// ID of associated trigger function:
  /// • 0: No Trigger (default): No trigger related behavior
  /// • >0: Trigger: o Start executing, when the trigger function with the identical EmitterID is triggered.
  /// Always positive.
  /// For more information, see chapter 5.5.12 Triggers
  ListenerID             : SINT;
  /// Reserve
  Reserve                : BYTE;
  /// Index of assigned conveyor
  ConveyorNo             : USINT;
  /// Relates to ListenerID >0
  /// Start index of real registers containing InitObjectPosition for trigger-based execution.
  StartIndexInitPosition : USINT;
  /// Relates to ListenerID = 0:
  /// Travel distance of assigned UCS between work piece detection (InitObjectPosition) and execution of this command.
  TrackingOffset         : REAL;
  /// Define the index number of the UCS that is assigned to the conveyor by the function "ConveyorTracking".
  /// For more information refer to chapter 5.5.14.
  FrameNo                : USINT;
  /// Relates to ListenerID >0
  /// Index of real register containing TrackingOffset for trigger-based execution
  IndexTrackingOffset    : USINT;
END_STRUCT
END_TYPE

{attribute 'pack_mode' := '1'} 
// ------------------------------------------------------------------------- 
//  SRCI Robot Library                                                
// ------------------------------------------------------------------------- 
//                                                                           
//  Object:      SyncToConveyorOutCmd                                       
//  Author:      Thorsten Brach                                                
//  Date:        2024-06-11
//
//  Description:                                              
//   
//                                                                           
//  Copyright: 
//    (C) 2024 Thorsten Brach. All rights reserved                                                                                                                                                                                                               
//             Licensed under the MIT License.
//                                                                           
//  Disclaimer:                                                                           
//    This project is provided without any guarantee and can be used for   
//    private and commercial purposes. Any use is at the user’s 
//    own risk and responsibility.
//
// -------------------------------------------------------------------------
TYPE SyncToConveyorOutCmd :
STRUCT
  /// Relates to ListenerID >0
  /// Number of successful trigger-based command invocations - For more information refer TO chapter 5.5.12.4
  InvocationCounter      : USINT;  
  /// Reserve
  Reserve                : BYTE;
  /// Unique system-generated ID of the "Action" when the function is triggered.
  /// • >0: The "Action" is started by the trigger funcrion with identical FollowID.
  /// • <0: The "Action" is stopped by the trigger function with identical FollowID.
  /// For more information see chapter 5.5.12.4 EmitterID, ListenerID, FollowID and OriginID
  OriginID               : INT;
  /// The TCP is in synchronization with the object on the conveyor belt.
  InSync                 : BOOL;
END_STRUCT
END_TYPE

{attribute 'pack_mode' := '1'} 
// ------------------------------------------------------------------------- 
//  SRCI Robot Library                                                
// ------------------------------------------------------------------------- 
//                                                                           
//  Object:      SyncToConveyorParCmd                                       
//  Author:      Thorsten Brach                                                
//  Date:        2024-06-11
//
//  Description:                                              
//   
//                                                                           
//  Copyright: 
//    (C) 2024 Thorsten Brach. All rights reserved                                                                                                                                      
//             Licensed under the MIT License.
//                                                                           
//  Disclaimer:                                                                           
//    This project is provided without any guarantee and can be used for   
//    private and commercial purposes. Any use is at the user’s 
//    own risk and responsibility.
//
// -------------------------------------------------------------------------
TYPE SyncToConveyorParCmd :
STRUCT
  /// Index of assigned conveyor
  ConveyorNo      : USINT;
  /// Define the index number of the UCS that will be assigned to the conveyor.
  /// For more information refer to chapter 5.5.14
  FrameNo         : USINT;
  /// Defines when synchronization starts.
  SyncInMode      : SyncInMode;
  /// Relates to "SyncInMode" "After distance" (1) and "After time" (2):
  /// Parameter for the synchronization
  /// • "After distance" (1)
  ///    •  Distance in mm
  /// • "After time" (2)
  ////   • Time in ms
  SyncInParameter : REAL;
  /// Define the maximum adjustment velocity for the robot to catch up to the conveyor belt.
  /// The velocity must be greater than the velocity of the conveyor belt.
  /// • 0 (default): no limit
  ///       o No conveyor tracking specific limit
  ///       o RC internal limit applies
  /// • >0: use limit
  ///       o Conveyor tracking specific limit applies
  MaxVelocity     : REAL;
  /// Define the maximum adjustment acceleration for the robot to catch up to the conveyor belt.
  /// • 0 (default): no limit
  ///     o No conveyor tracking specific limit
  ///     o RC internal limit applies
  /// • >0: use limit
  ///     o Conveyor tracking specific limit applies
  MaxAcceleration : REAL;
  /// ID of associated trigger function:
  ///  •  0: No Trigger (default):
  ///        o No trigger related behavior
  ///  • >0: Trigger:
  ///        o Start executing, when the trigger function with the identical EmitterID is triggered.
  /// Always positive.
  /// For more information, see chapter 5.5.12 Triggers
  ListenerID      : SINT;
END_STRUCT
END_TYPE

{attribute 'pack_mode' := '1'} 
// ------------------------------------------------------------------------- 
//  SRCI Robot Library                                                
// ------------------------------------------------------------------------- 
//                                                                           
//  Object:      SyncToConveyorRecvData                                       
//  Author:      Thorsten Brach                                                
//  Date:        2024-06-11
//
//  Description:                                              
//   
//                                                                           
//  Copyright: 
//    (C) 2024 Thorsten Brach. All rights reserved                                                                                                                                            
//             Licensed under the MIT License.
//                                                                           
//  Disclaimer:                                                                           
//    This project is provided without any guarantee and can be used for   
//    private and commercial purposes. Any use is at the user’s 
//    own risk and responsibility.
//
// -------------------------------------------------------------------------
TYPE SyncToConveyorRecvData EXTENDS RspHeader :
STRUCT
  InvocationCounter : USINT;
  /// Reserve
  Reserved          : SINT;
  /// Unique system-generated ID of the "Action" when the function is triggered.
  /// • >0: The "Action" is started by the trigger funcrion with identical FollowID.
  /// • <0: The "Action" is stopped by the trigger function with identical FollowID.
  /// For more information see chapter 5.5.12.4 EmitterID, ListenerID, FollowID and OriginID
  OriginID          : INT;
  /// The TCP is in synchronization with the object on the conveyor belt.
  InSync            : BOOL;
END_STRUCT
END_TYPE

{attribute 'pack_mode' := '1'}
// ------------------------------------------------------------------------- 
//  SRCI Robot Library                                                
// ------------------------------------------------------------------------- 
//                                                                           
//  Object:      SyncToConveyorSendData                                       
//  Author:      Thorsten Brach                                                
//  Date:        2024-06-11
//
//  Description:                                              
//   
//                                                                           
//  Copyright: 
//    (C) 2024 Thorsten Brach. All rights reserved                                                                                                                                            
//             Licensed under the MIT License.
//                                                                           
//  Disclaimer:                                                                           
//    This project is provided without any guarantee and can be used for   
//    private and commercial purposes. Any use is at the user’s 
//    own risk and responsibility.
//
// -------------------------------------------------------------------------
TYPE SyncToConveyorSendData EXTENDS CmdHeader:   
STRUCT
  /// EmitterID
  EmitterID       : ARRAY[0..3] OF SINT;
  /// ID of associated trigger function:
  /// • 0: No Trigger (default): No trigger related behavior
  /// • >0: Trigger: o Start executing, when the trigger function with the identical EmitterID is triggered.
  /// Always positive.
  /// For more information, see chapter 5.5.12 Triggers
  ListenerID      : SINT;
  /// Reserve
  Reserve         : BYTE;
  /// Index of assigned conveyor
  ConveyorNo      : USINT;
  /// Define the index number of the UCS that will be assigned to the conveyor.
  /// For more information refer to chapter 5.5.14
  FrameNo         : USINT;
  /// Defines when synchronization starts
  SyncInMode      : SyncInMode;
  /// Relates to "SyncInMode" "After distance" (1) and "After time" (2): Parameter for the synchronization
  /// • "After distance" (1) -  Distance in mm
  /// • "After time" (2) -  Time in ms
  SyncInParameter : REAL;
  /// Define the maximum adjustment velocity for the robot to catch up to the conveyor belt.
  /// The velocity must be greater than the velocity of the conveyor belt.
  /// • 0 (default): no limit - No conveyor tracking specific limit
  ///                         - RC internal limit applies
  /// • >0: use limit         - Conveyor tracking specific limit applies
  MaxVelocity     : REAL;
  /// Define the maximum adjustment acceleration for the robot to catch up to the conveyor belt.
  /// • 0 (default): no limit - No conveyor tracking specific limit
  ///                         - RC internal limit applies
  /// • >0: use limit         - Conveyor tracking specific limit applies
  MaxAcceleration : REAL;
  /// ID of associated trigger function:
  /// • 0: No Trigger (default): No trigger related behavior
  /// • >0: Trigger:  Start executing, when the trigger function with the identical EmitterID is triggered.
  /// Always positive.
  /// For more information, see chapter 5.5.12 Triggers
END_STRUCT
END_TYPE

{attribute 'pack_mode' := '1'} 
// ------------------------------------------------------------------------- 
//  SRCI Robot Library                                                
// ------------------------------------------------------------------------- 
//                                                                           
//  Object:      ForceControlOutCmd                                       
//  Author:      Thorsten Brach                                                
//  Date:        2024-06-16
//
//  Description:                                              
//   
//                                                                           
//  Copyright: 
//    (C) 2024 Thorsten Brach. All rights reserved                                                                                                                                                                                                               
//             Licensed under the MIT License.
//                                                                           
//  Disclaimer:                                                                           
//    This project is provided without any guarantee and can be used for   
//    private and commercial purposes. Any use is at the user’s 
//    own risk and responsibility.
//
// -------------------------------------------------------------------------
TYPE ForceControlOutCmd :
STRUCT
  /// Current status of ForceControl and ForceLimit (chapter 6.5.25) according to Table 6-712
  ForceStatus        : ForceStatus;  
END_STRUCT
END_TYPE

{attribute 'pack_mode' := '1'} 
// ------------------------------------------------------------------------- 
//  SRCI Robot Library                                                
// ------------------------------------------------------------------------- 
//                                                                           
//  Object:      ForceControlParCmd                                       
//  Author:      Thorsten Brach                                                
//  Date:        2024-06-16
//
//  Description:                                              
//   
//                                                                           
//  Copyright: 
//    (C) 2024 Thorsten Brach. All rights reserved                                                                                                                                      
//             Licensed under the MIT License.
//                                                                           
//  Disclaimer:                                                                           
//    This project is provided without any guarantee and can be used for   
//    private and commercial purposes. Any use is at the user’s 
//    own risk and responsibility.
//
// -------------------------------------------------------------------------
TYPE ForceControlParCmd :
STRUCT
  /// Defines type of reference of Force and Torque (at least one option must be supported)
  ReferenceType      : ReferenceType;
  /// Relates to ConnectionMode 1 and 2 (Sensor connected to PLC).
  /// Currently applied force and torque detected by sensor according to ReferenceType, ToolNo and FrameNo.
  /// • [0]: X-Axis
  /// • [1]: Y-Axis
  /// • [2]: Z- Axis
  /// • [3]: Rotation around X-Axis (RX)
  /// • [4]: Rotation around Y-Axis (RY)
  /// • [5]: Rotation around Z- Axis (RZ)
  SensorValue        : ARRAY[0..5] OF REAL;
  /// Relates to ReferenceType 0 (Tool) and 1 (Frame):
  /// Force and torque to be applied by robot arm according to ReferenceType, ToolNo and FrameNo:
  /// • [0]: X-Axis
  /// • [1]: Y-Axis
  /// • [2]: Z- Axis
  /// • [3]: Rotation around X-Axis (RX)
  /// • [4]: Rotation around Y-Axis (RY)
  /// • [5]: Rotation around Z- Axis (RZ)
  /// Set TargetValue <>-99999.9999 (default) to define setpoint
  TargetValue        : ARRAY[0..5] OF REAL;
  /// Index of tool
  /// •      0: Flange (default)
  /// • 1..254: Tool frames
  ToolNo             : USINT;
  /// Define the index number of the UCS that will be assigned to the conveyor.
  /// For more information refer to chapter 5.5.14
  FrameNo            : USINT;
  /// Specifies encoder connection setup according to Table 6-713 (at least one option must be supported) 
  ConnectionMode     : SensorConnectionMode;
  /// Position of sensor relative to flange (FixedSensor FALSE) or relative to WCS (FixedSensor TRUE)
  /// • [0]: X-Axis
  /// • [1]: Y-Axis
  /// • [2]: Z- Axis
  /// • [3]: Rotation around X-Axis (RX)
  /// • [4]: Rotation around Y-Axis (RY)
  /// • [5]: Rotation around Z- Axis (RZ)
  SensorFrame        : ARRAY[0..5] OF REAL;
  /// Index of payload data containing mass, center of gravity, orientation and inertia relative to SensorFrame.
  /// Required to calibrate system for setting up gravity compensation and sensor offset.
  CalibrationData    : USINT;
  /// Tolerance of TargetValue within which currently applied force/torque will return ForceStatus "Specified force/torque reached" TRUE.
  TargetWindow       : REAL;
  /// Define axes whose position may be adjusted by the robot to apply specified force according to Table 6-711.
  CompliantAxes      : BYTE;
  /// Maximum allowed TCP velocity for compliant axes in % of nominal velocity.
  /// •   0% (default): no limit - RC internal limit applies
  /// •  >0% use limit -  Specified limit applies
  /// • 100% use maximal reference velocity
  /// For more information on nominal dynamics see chapter 5.5.7 Robot dynamics 
  MaxVelocity        : UINT;
  /// Maximum allowed cartesian deviation according to ReferenceType, ToolNo and FrameNo.
  /// Set 0 (default) to not specify a limit in this axis direction.
  /// • [0]: Deviation in X-Direction in mm
  /// • [1]: Deviation in Y- direction in mm
  /// • [2]: Deviation in Z- direction in mm
  /// • [3]: Deviation in RX- direction in °
  /// • [4]: Deviation in RY- direction in °
  /// • [5]: Deviation in RZ- direction in °
  MaxDeviation       : ARRAY [0..5] OF REAL;
  /// Defines reaction in case ForceControl reports error during its execution
  /// Processing of active move command is continued without active ForceControl
  ErrorReaction      : ErrorReaction;
  /// Relates to ErrorReaction 0 (Abort and move). Defines type of reference coordinate system of ErrorVector
  ErrorReferenceType : ReferenceType;
  /// Relates to ErrorReaction 0 (Abort and move). Vector defining robot’s movement in case of
  /// incoming error according to ErrorReferenceType, ErrorToolNo and ErrorFrameNo.
  /// • [0]: X-Axis
  /// • [1]: Y-Axis
  /// • [2]: Z- Axis
  /// • [3]: Rotation around X-Axis (RX)
  /// • [4]: Rotation around Y-Axis (RY)
  /// • [5]: Rotation around Z-Axis (RZ)
  ErrorVector        : ARRAY [0..5] OF REAL;
  /// Relates to ErrorReaction 0 (Abort and move). Index of tool.
  /// • 0 (default): Flange
  /// • 1..254: Tool frames
  ErrorToolNo        : USINT;
  /// Relates to ErrorReferenceType 1 (Frame)
  /// •      0: WCS (default)
  /// • 1..254: User frames
  ErrorFrameNo       : USINT;
  /// Defines sensor positioning:
  /// • FALSE (default): Sensor mounted on flange
  /// • TRUE: Sensor fixed
  FixedSensor        : BOOL;
END_STRUCT
END_TYPE

{attribute 'pack_mode' := '1'} 
// ------------------------------------------------------------------------- 
//  SRCI Robot Library                                                
// ------------------------------------------------------------------------- 
//                                                                           
//  Object:      ForceControlRecvData                                       
//  Author:      Thorsten Brach                                                
//  Date:        2024-06-11
//
//  Description:                                              
//   
//                                                                           
//  Copyright: 
//    (C) 2024 Thorsten Brach. All rights reserved                                                                                                                                            
//             Licensed under the MIT License.
//                                                                           
//  Disclaimer:                                                                           
//    This project is provided without any guarantee and can be used for   
//    private and commercial purposes. Any use is at the user’s 
//    own risk and responsibility.
//
// -------------------------------------------------------------------------
TYPE ForceControlRecvData EXTENDS RspHeader :
STRUCT
  /// Current status of ForceControl and ForceLimit (chapter 6.5.25) according to Table 6-712
  ForceStatus : BYTE;
END_STRUCT
END_TYPE

{attribute 'pack_mode' := '1'}
// ------------------------------------------------------------------------- 
//  SRCI Robot Library                                                
// ------------------------------------------------------------------------- 
//                                                                           
//  Object:      ForceControlSendData                                       
//  Author:      Thorsten Brach                                                
//  Date:        2024-06-11
//
//  Description:                                              
//   
//                                                                           
//  Copyright: 
//    (C) 2024 Thorsten Brach. All rights reserved                                                                                                                                            
//             Licensed under the MIT License.
//                                                                           
//  Disclaimer:                                                                           
//    This project is provided without any guarantee and can be used for   
//    private and commercial purposes. Any use is at the user’s 
//    own risk and responsibility.
//
// -------------------------------------------------------------------------
TYPE ForceControlSendData EXTENDS CmdHeader:   
STRUCT
  /// Index of tool
  /// •      0: Flange (default)
  /// • 1..254: Tool frames
  ToolNo             : USINT;
  /// Define the index number of the UCS that will be assigned to the conveyor.
  /// For more information refer to chapter 5.5.14
  FrameNo            : USINT;
  /// Specifies encoder connection setup according to Table 6-713 (at least one option must be supported) 
  ConnectionMode     : SensorConnectionMode;
  /// Defines sensor positioning:
  /// • FALSE (default): Sensor mounted on flange
  /// • TRUE: Sensor fixed
  FixedSensor        : BYTE;
  /// Position of sensor relative to flange (FixedSensor FALSE) or relative to WCS (FixedSensor TRUE)
  /// • [0]: X-Axis
  /// • [1]: Y-Axis
  /// • [2]: Z- Axis
  /// • [3]: Rotation around X-Axis (RX)
  /// • [4]: Rotation around Y-Axis (RY)
  /// • [5]: Rotation around Z- Axis (RZ)
  SensorFrame        : ARRAY[0..5] OF REAL;
  /// Index of payload data containing mass, center of gravity, orientation and inertia relative to SensorFrame.
  /// Required to calibrate system for setting up gravity compensation and sensor offset.
  CalibrationData    : USINT;
  /// Defines type of reference of Force and Torque (at least one option must be supported)
  ReferenceType      : ReferenceType;
  /// Relates to ConnectionMode 1 and 2 (Sensor connected to PLC).
  /// Currently applied force and torque detected by sensor according to ReferenceType, ToolNo and FrameNo.
  /// • [0]: X-Axis
  /// • [1]: Y-Axis
  /// • [2]: Z- Axis
  /// • [3]: Rotation around X-Axis (RX)
  /// • [4]: Rotation around Y-Axis (RY)
  /// • [5]: Rotation around Z- Axis (RZ)
  SensorValue        : ARRAY[0..5] OF REAL;
  /// Relates to ReferenceType 0 (Tool) and 1 (Frame):
  /// Force and torque to be applied by robot arm according to ReferenceType, ToolNo and FrameNo:
  /// • [0]: X-Axis
  /// • [1]: Y-Axis
  /// • [2]: Z- Axis
  /// • [3]: Rotation around X-Axis (RX)
  /// • [4]: Rotation around Y-Axis (RY)
  /// • [5]: Rotation around Z- Axis (RZ)
  /// Set TargetValue <>-99999.9999 (default) to define setpoint
  TargetValue        : ARRAY[0..5] OF REAL;
  /// Maximum allowed TCP velocity for compliant axes in % of nominal velocity.
  /// •   0% (default): no limit - RC internal limit applies
  /// •  >0% use limit -  Specified limit applies
  /// • 100% use maximal reference velocity
  /// For more information on nominal dynamics see chapter 5.5.7 Robot dynamics 
  MaxVelocity        : UINT;
  /// Maximum allowed cartesian deviation according to ReferenceType, ToolNo and FrameNo.
  /// Set 0 (default) to not specify a limit in this axis direction.
  /// • [0]: Deviation in X-Direction in mm
  /// • [1]: Deviation in Y- direction in mm
  /// • [2]: Deviation in Z- direction in mm
  /// • [3]: Deviation in RX- direction in °
  /// • [4]: Deviation in RY- direction in °
  /// • [5]: Deviation in RZ- direction in °
  MaxDeviation       : ARRAY [0..5] OF REAL;
  /// Defines reaction in case ForceControl reports error during its execution
  /// Processing of active move command is continued without active ForceControl
  ErrorReaction      : ErrorReaction;
  /// Relates to ErrorReaction 0 (Abort and move). Defines type of reference coordinate system of ErrorVector
  ErrorReferenceType : ReferenceType;
  /// Relates to ErrorReaction 0 (Abort and move). Vector defining robot’s movement in case of
  /// incoming error according to ErrorReferenceType, ErrorToolNo and ErrorFrameNo.
  /// • [0]: X-Axis
  /// • [1]: Y-Axis
  /// • [2]: Z- Axis
  /// • [3]: Rotation around X-Axis (RX)
  /// • [4]: Rotation around Y-Axis (RY)
  /// • [5]: Rotation around Z-Axis (RZ)
  ErrorVector        : ARRAY [0..5] OF REAL;
  /// Relates to ErrorReaction 0 (Abort and move). Index of tool.
  /// • 0 (default): Flange
  /// • 1..254: Tool frames
  ErrorToolNo        : USINT;
  /// Relates to ErrorReferenceType 1 (Frame)
  /// •      0: WCS (default)
  /// • 1..254: User frames
  ErrorFrameNo       : USINT;
  /// Define axes whose position may be adjusted by the robot to apply specified force according to Table 6-711.
  CompliantAxes      : BYTE;
END_STRUCT
END_TYPE

